ABB RobotStudio station: SD_RStudioExe01_240509.rsstnx

Station SD_RStudioExe01_240509 (saved by RobotStudio 22.3.10190.2)
Controller CRB15000_5_95_1
  mechanical unit ROB_1: CRB15000_5_95__02, 6 joints, base frame (0, 0, 0) mm
Layout (positions relative to the parent item):
  - CRB15000_5_95__02 [mechanism, from Robots\CRB15000_5_95__02.rslib] at (0, 0, 0) mm; joint values [0.5369, -0.3436, 0.8085, -0.0017, 0.992, 2.564] (rad or m)
  - SD_UteCono [mechanism] at (353.07, 210.07, 479.41) mm, rotated rx 176.35 ry -5.42 rz 64.08 deg
      TCP SD_UteCono at (0, 0, 80) mm
      links: Parte_1
  - Parte_1 [part] at (360.49, 214.63, 0) mm, size 300 x 300 x 400 mm
Attachment: SD_UteCono is attached to CRB15000_5_95__02 / Link6
Targets, tools, work objects and paths stored in the station, written as RAPID:
! task T_ROB1
MODULE CalibData
  PERS tooldata SD_UteCono:=[TRUE,[[0,0,80],[1,0,0,0]],[1,[0,0,1],[1,0,0,0],0,0,0]];
  PERS wobjdata Workobject_2:=[FALSE,TRUE,"",[[360.491,214.626,400],[0,0,1,0]],[[0,0,0],[1,0,0,0]]];
ENDMODULE

! task T_ROB1
MODULE Module1
  CONST robtarget Target_10:=[[-299.99985192,0.36769812,0],[0.707106781,0,0,0.707106781],[0,0,0,0],[9E+09,9E+09,9E+09,9E+09,9E+09,9E+09]];
  CONST robtarget Target_20:=[[-0.447873291,0.000329183,0],[0,0,0.707106781,0.707106781],[0,1,1,0],[9E+09,9E+09,9E+09,9E+09,9E+09,9E+09]];
  PROC Path_10()
    MoveJ Target_10,v1000,z100,SD_UteCono\WObj:=Workobject_2;
    MoveJ Target_20,v1000,z100,SD_UteCono\WObj:=Workobject_2;
  ENDPROC
ENDMODULE

